(* CoDeSys 2.3 export: VARIABLE_CONFIGURATION.EXP *)

(* Global variable list: Variable_Configuration *)
VAR_GLOBAL RETAIN
	K14UZSPumpSpeed : USINT := 100;
END_VAR
